// TIA Portal V17 export
// export: Created 2024-09-02T12:50:29.3841235Z, ExportSetting WithDefaults, DisplayName Totally Integrated Automation Portal, DisplayVersion V17, DisplayName TIA Portal Openness, DisplayVersion V17, DisplayName TIA Portal Version Control Interface, DisplayVersion V17, DisplayName STEP 7 Professional, DisplayVersion V17, DisplayName STEP 7 Safety, DisplayVersion V17, DisplayName WinCC Professional, DisplayVersion V17
TYPE "TypeDirektstarter_out"
// stored: IsFailsafeCompliant false
   STRUCT
      MotorOnLeft : Bool;   // Motor Linkslauf ein / Motor left rotation on
      MotorOnRight : Bool;   // Motor Rechtslauf ein / Motor clockwise rotation on
      Break : Bool;   // Ansteuerung für Bremse / Control for brake
      Reset : Bool;   // Trip-Reset / Trip reset
      Emergency : Bool;   // Notstart / emergency start
      Selftest : Bool;   // Selbsttest / Self test
      res07 : Bool;   // n.c.
      res08 : Bool;   // n.c.
      res09 : Bool;   // n.c.
      res10 : Bool;   // n.c.
      res11 : Bool;   // n.c.
      res12 : Bool;   // n.c.
      res13 : Bool;   // n.c.
      res14 : Bool;   // n.c.
      res15 : Bool;   // n.c.
      QuickStopLocked : Bool;   // Quick-Stop sperren / Lock Quick-Stop
   END_STRUCT;
END_TYPE
